FUNCTION FC_StartStopReset : BOOL
VAR_INPUT
END_VAR
VAR
END_VAR

// start/stopknop regeling
IF (DB10_Alias.ix_stopKnop AND DB10_Alias.ix_startKnop) OR NOT GVL.safetyOK THEN
	DB_PRG1.PRG1Stap := 950;	 

ELSIF DB10_Alias.ix_stopKnop THEN
	GVL.b_StopPRG := TRUE;
	GVL.b_StartPRG := FALSE;
ELSIF DB10_Alias.ix_startKnop THEN
	GVL.b_StartPRG := TRUE;
	GVL.b_StopPRG := FALSE;
END_IF

END_FUNCTION

(* stored: Version 1.1.0.1, ProductVersion 3.1.4024.12
   POU FC_StartStopReset: Id {dee57a70-d1bc-45b5-be67-c879719edd13}, SpecialFunc None *)
